// Library/Structures/Miscellaneous/RCSupportedFunctions
{attribute 'pack_mode' := '1'} 
// ------------------------------------------------------------------------- 
//  SRCI Robot Library                                                
// ------------------------------------------------------------------------- 
//                                                                           
//  Object:      RCSupportedFunctions                                       
//  Author:      Thorsten Brach                                                
//  Date:        2024-06-01
//
//  Description:                                              
//   
//                                                                           
//  Copyright: 
//    (C) 2024 Thorsten Brach. All rights reserved                                                                                                                                            
//             Licensed under the LGPL-3.0 license.
//                                                                           
//  Disclaimer:                                                                           
//    This project is provided without any guarantee and can be used for   
//    private and commercial purposes. Any use is at the user’s 
//    own risk and responsibility.
//
// -------------------------------------------------------------------------
TYPE RCSupportedFunctions :
STRUCT
  /// Byte 00 - Bit 0  
  Reserved                   : BOOL;
  /// Byte 00 - Bit 1 -> must be initialized with true, because this command is part of the interface initialization
  ReadRobotData              : BOOL := TRUE; 
  /// Byte 00 - Bit 2  
  EnableRobot                : BOOL;
  /// Byte 00 - Bit 3  
  GroupReset                 : BOOL;
  /// Byte 00 - Bit 4  
  ReadActualPosition         : BOOL;
  /// Byte 00 - Bit 5 
  ReadActualPositionCyclic   : BOOL;
  /// Byte 00 - Bit 6  -> must be initialized with true, because this command is part of the interface initialization
  ExchangeConfiguration      : BOOL := TRUE; 
  /// Byte 00 - Bit 7  
  SetSequence                : BOOL;
  
  /// Byte 01 - Bit 0  
  ChangeSpeedOverride        : BOOL;
  /// Byte 01 - Bit 1  ->  must be initialized with true, because this command is part of the interface initialization
  ReadMessages               : BOOL := TRUE; 
  /// Byte 01 - Bit 2  
  ReadRobotReferenceDynamics : BOOL;
  /// Byte 01 - Bit 3  
  WriteFrameData             : BOOL;
  /// Byte 01 - Bit 4  
  WriteToolData              : BOOL;
  /// Byte 01 - Bit 5  
  WriteLoadData              : BOOL;
  /// Byte 01 - Bit 6  
  WriteRobotReferenceDynamics: BOOL;
  /// Byte 01 - Bit 7  
  WriteRobotDefaultDynamics  : BOOL;
  
  /// Byte 02 - Bit 0  
  ReadRobotDefaultDynamics   : BOOL;
  /// Byte 02 - Bit 1  
  ReadFrameData              : BOOL;
  /// Byte 02 - Bit 2  
  ReadToolData               : BOOL;
  /// Byte 02 - Bit 3  
  ReadLoadData               : BOOL;
  /// Byte 02 - Bit 4  
  ReadRobotSWLimits          : BOOL;
  /// Byte 02 - Bit 5  
  GroupJog                   : BOOL;
  /// Byte 02 - Bit 6  
  MoveLinearAbsolute         : BOOL;
  /// Byte 02 - Bit 7  
  MoveDirectAbsolute         : BOOL;
  
  /// Byte 03 - Bit 0  
  MoveAxesAbsolute           : BOOL;
  /// Byte 03 - Bit 1  
  GroupStop                  : BOOL;
  /// Byte 03 - Bit 2
  GroupContinue              : BOOL;
  /// Byte 03 - Bit 3
  GroupInterrupt             : BOOL;
  /// Byte 03 - Bit 4
  ReturnToPrimary            : BOOL;
  /// Byte 03 - Bit 5
  MoveLinearAbsoluteJ        : BOOL;
  /// Byte 03 - Bit 6
  MoveDirectRelative         : BOOL;
  /// Byte 03 - Bit 7
  MoveAxesRelative           : BOOL;
  
  /// Byte 04 - Bit 0
  MoveCircularAbsolute       : BOOL;
  /// Byte 04 - Bit 1
  MoveCircularRelative       : BOOL;
  /// Byte 04 - Bit 2
  MoveLinearOffset           : BOOL;
  /// Byte 04 - Bit 3
  MoveDirectOffset           : BOOL;
  /// Byte 04 - Bit 4
  WaitTime                   : BOOL;
  /// Byte 04 - Bit 5
  ReadDigitalInputs          : BOOL;
  /// Byte 04 - Bit 6
  ReadDigitalOutputs         : BOOL;
  /// Byte 04 - Bit 7
  WriteDigitalOutputs        : BOOL;
  
  /// Byte 05 - Bit 0
  ReadIntegers               : BOOL;
  /// Byte 05 - Bit 1
  ReadReals                  : BOOL;
  /// Byte 05 - Bit 2
  WriteIntegers              : BOOL;
  /// Byte 05 - Bit 3
  WriteReals                 : BOOL;
  /// Byte 05 - Bit 4
  MoveLinearCam              : BOOL;
  /// Byte 05 - Bit 5
  MoveDirectCam              : BOOL;
  /// Byte 05 - Bit 6
  MoveCircularCam            : BOOL;
  /// Byte 05 - Bit 7
  SetTriggerRegister         : BOOL;
  
  /// Byte 06 - Bit 0
  SetTriggerLimit            : BOOL;
  /// Byte 06 - Bit 1
  SetTriggerUser             : BOOL;
  /// Byte 06 - Bit 2
  SetTriggerError            : BOOL;
  /// Byte 06 - Bit 3
  ReactAtTrigger             : BOOL;
  /// Byte 06 - Bit 4
  WaitForTrigger             : BOOL;
  /// Byte 06 - Bit 5
  ReadSystemVariable         : BOOL;
  /// Byte 06 - Bit 6
  WriteSystemVariable        : BOOL;
  /// Byte 06 - Bit 7
  CalculateForwardKinematic  : BOOL;
  
  /// Byte 07 - Bit 0
  CalculateInverseKinematic  : BOOL;
  /// Byte 07 - Bit 1
  CalculateCartesianPosition : BOOL;
  /// Byte 07 - Bit 2
  CalculateTool              : BOOL;
  /// Byte 07 - Bit 3
  CalculateFrame             : BOOL;
  /// Byte 07 - Bit 4
  ActivateNextCommand        : BOOL;
  /// Byte 07 - Bit 5
  ShiftPosition              : BOOL;
  /// Byte 07 - Bit 6
  CallSubprogram             : BOOL;
  /// Byte 07 - Bit 7
  MoveLinearRelative         : BOOL;
  
  /// Byte 08 - Bit 0
  WriteCallSubprogramCyclic  : BOOL;
  /// Byte 08 - Bit 1
  ReadCallSubprogramCyclic   : BOOL;
  /// Byte 08 - Bit 2
  StopSubprogram             : BOOL;
  /// Byte 08 - Bit 3
  ReadDHParameter            : BOOL;
  /// Byte 08 - Bit 4
  RestartController          : BOOL;
  /// Byte 08 - Bit 5
  ReadActualTCPVelocity      : BOOL;
  /// Byte 08 - Bit 6
  UserLogin                  : BOOL;
  /// Byte 08 - Bit 7
  SwitchLanguage             : BOOL;
  
  /// Byte 09 - Bit 0
  WriteRobotSWLimits         : BOOL;
  /// Byte 09 - Bit 1
  SetOperationMode           : BOOL;
  /// Byte 09 - Bit 2
  ReadWorkArea               : BOOL;
  /// Byte 09 - Bit 3
  WriteWorkArea              : BOOL;
  /// Byte 09 - Bit 4
  ActivateWorkArea           : BOOL;
  /// Byte 09 - Bit 5
  MonitorWorkArea            : BOOL;
  /// Byte 09 - Bit 6
  MoveApproachLinear         : BOOL;
  /// Byte 09 - Bit 7
  MoveDepartLinear           : BOOL;
  
  /// Byte 10 - Bit 0
  MoveApproachDirect         : BOOL;
  /// Byte 10 - Bit 1
  MoveDepartDirect           : BOOL;
  /// Byte 10 - Bit 2
  SearchHardstop             : BOOL;
  /// Byte 10 - Bit 3
  SearchHardstopJ            : BOOL;
  /// Byte 10 - Bit 4
  MovePickPlaceLinear        : BOOL;
  /// Byte 10 - Bit 5
  MovePickPlaceDirect        : BOOL;
  /// Byte 10 - Bit 6
  ActivateConveyorTracking   : BOOL;
  /// Byte 10 - Bit 7
  RedefineTrackingPosition   : BOOL;

  /// Byte 11 - Bit 0
  SyncToConveyor             : BOOL;
  /// Byte 11 - Bit 1
  ConfigureConveyor          : BOOL;
  /// Byte 11 - Bit 2
  MoveSuperImposed           : BOOL;
  /// Byte 11 - Bit 3
  MoveSuperImposedDynamic    : BOOL;
  /// Byte 11 - Bit 4
  ReadAnalogInput            : BOOL;
  /// Byte 11 - Bit 5
  ReadAnalogOutput           : BOOL;
  /// Byte 11 - Bit 6
  WriteAnalogOutput          : BOOL;
  /// Byte 11 - Bit 7
  MeasuringInput             : BOOL;

  /// Byte 12 - Bit 0
  AbortMeasuringInput        : BOOL;
  /// Byte 12 - Bit 1
  SetTriggerMotion           : BOOL;
  /// Byte 12 - Bit 2
  OpenBrake                  : BOOL;
  /// Byte 12 - Bit 3
  PathAccuracyMode           : BOOL;
  /// Byte 12 - Bit 4
  AvoidSingularity           : BOOL;
  /// Byte 12 - Bit 5
  ForceControl               : BOOL;
  /// Byte 12 - Bit 6
  ForceLimit                 : BOOL;
  /// Byte 12 - Bit 7
  ReadActualForce            : BOOL;
  
  /// Byte 13 - Bit 0
  BrakeTest                  : BOOL;
  /// Byte 13 - Bit 1
  SoftSwitchTCP              : BOOL;
  /// Byte 13 - Bit 2
  CreateSpline               : BOOL;
  /// Byte 13 - Bit 3
  DeleteSpline               : BOOL;
  /// Byte 13 - Bit 4
  MoveSpline                 : BOOL;
  /// Byte 13 - Bit 5
  DynamicSpline              : BOOL;
  /// Byte 13 - Bit 6
  LoadMeasurementAutomatic   : BOOL;
  /// Byte 13 - Bit 7
  LoadMeasurementSequential  : BOOL;
  
  /// Byte 14 - Bit 0
  CollisionDetection         : BOOL;
  /// Byte 14 - Bit 1
  FreeDrive                  : BOOL;
  /// Byte 14 - Bit 2
  UnitMeasurement            : BOOL;
  /// Byte 14 - Bit 3
  Byte14Bit03                : BOOL;
  /// Byte 14 - Bit 4
  Byte14Bit04                : BOOL;
  /// Byte 14 - Bit 5
  Byte14Bit05                : BOOL;
  /// Byte 14 - Bit 6
  Byte14Bit06                : BOOL;
  /// Byte 14 - Bit 7
  Byte14Bit07                : BOOL;
  
  /// Byte 15 - Bit 0
  Byte15Bit00                : BOOL;
  /// Byte 15 - Bit 1
  Byte15Bit01                : BOOL;
  /// Byte 15 - Bit 2
  Byte15Bit02                : BOOL;
  /// Byte 15 - Bit 3
  Byte15Bit03                : BOOL;
  /// Byte 15 - Bit 4
  Byte15Bit04                : BOOL;
  /// Byte 15 - Bit 5
  Byte15Bit05                : BOOL;
  /// Byte 15 - Bit 6
  Byte15Bit06                : BOOL;
  /// Byte 15 - Bit 7
  Byte15Bit07                : BOOL;

  /// Byte 16 - Bit 0
  Byte16Bit00                : BOOL;
  /// Byte 15 - Bit 1
  Byte16Bit01                : BOOL;
  /// Byte 15 - Bit 2
  Byte16Bit02                : BOOL;
  /// Byte 15 - Bit 3
  Byte16Bit03                : BOOL;
  /// Byte 15 - Bit 4
  Byte16Bit04                : BOOL;
  /// Byte 15 - Bit 5
  Byte16Bit05                : BOOL;
  /// Byte 15 - Bit 6
  Byte16Bit06                : BOOL;
  /// Byte 15 - Bit 7
  Byte16Bit07                : BOOL;
  
  /// Byte 17 - Bit 0
  Byte17Bit00                : BOOL;
  /// Byte 17 - Bit 1
  Byte17Bit01                : BOOL;
  /// Byte 17 - Bit 2
  Byte17Bit02                : BOOL;
  /// Byte 17 - Bit 3
  Byte17Bit03                : BOOL;
  /// Byte 17 - Bit 4
  Byte17Bit04                : BOOL;
  /// Byte 17 - Bit 5
  Byte17Bit05                : BOOL;
  /// Byte 17 - Bit 6
  Byte17Bit06                : BOOL;
  /// Byte 17 - Bit 7
  Byte17Bit07                : BOOL;

  /// Byte 18 - Bit 0
  Byte18Bit00                : BOOL;
  /// Byte 18 - Bit 1
  Byte18Bit01                : BOOL;
  /// Byte 18 - Bit 2
  Byte18Bit02                : BOOL;
  /// Byte 18 - Bit 3
  Byte18Bit03                : BOOL;
  /// Byte 18 - Bit 4
  Byte18Bit04                : BOOL;
  /// Byte 18 - Bit 5
  Byte18Bit05                : BOOL;
  /// Byte 18 - Bit 6
  Byte18Bit06                : BOOL;
  /// Byte 18 - Bit 7
  Byte18Bit07                : BOOL;
END_STRUCT
END_TYPE

// Library/Structures/Miscellaneous/RobotAxesFlags
{attribute 'pack_mode' := '1'} 
// ------------------------------------------------------------------------- 
//  SRCI Robot Library                                                
// ------------------------------------------------------------------------- 
//                                                                           
//  Object:      RobotAxesFlags                                       
//  Author:      Thorsten Brach                                                
//  Date:        2024-06-01
//
//  Description:                                              
//   
//                                                                           
//  Copyright: 
//    (C) 2024 Thorsten Brach. All rights reserved                                                                                                                                            
//             Licensed under the LGPL-3.0 license.
//                                                                           
//  Disclaimer:                                                                           
//    This project is provided without any guarantee and can be used for   
//    private and commercial purposes. Any use is at the user’s 
//    own risk and responsibility.
//
// -------------------------------------------------------------------------
TYPE RobotAxesFlags :
STRUCT
  /// Bit00 : Not used
  Bit00   : BOOL;
  /// Bit01 : Robot axis J1 - property depends of usage 
  AxisJ1  : BOOL;
  /// Bit02 : Robot axis J2 - property depends of usage 
  AxisJ2  : BOOL;
  /// Bit03 : Robot axis J3 - property depends of usage 
  AxisJ3  : BOOL;
  /// Bit04 : Robot axis J4 - property depends of usage 
  AxisJ4  : BOOL;
  /// Bit05 : Robot axis J5 - property depends of usage 
  AxisJ5  : BOOL;
  /// Bit06 : Robot axis J6 - property depends of usage 
  AxisJ6  : BOOL;
  /// Bit07 : Not used
  Bit07   : BOOL;
END_STRUCT
END_TYPE

// Library/Structures/Miscellaneous/SWLimits
{attribute 'pack_mode' := '1'} 
// ------------------------------------------------------------------------- 
//  SRCI Robot Library                                                
// ------------------------------------------------------------------------- 
//                                                                           
//  Object:      SWLimits                                       
//  Author:      Thorsten Brach                                                
//  Date:        2024-06-01
//
//  Description:                                              
//   
//                                                                           
//  Copyright: 
//    (C) 2024 Thorsten Brach. All rights reserved                                                                                                                                            
//             Licensed under the LGPL-3.0 license.
//                                                                           
//  Disclaimer:                                                                           
//    This project is provided without any guarantee and can be used for   
//    private and commercial purposes. Any use is at the user’s 
//    own risk and responsibility.
//
// -------------------------------------------------------------------------
TYPE SWLimits :
STRUCT
  /// Timestamp
  Timestamp    : IEC_TIMESTAMP;
  /// Negative software limit for Joint J1 [mm/°]
  J1LowerLimit : REAL;
  /// Positive software limit for Joint J1 [mm/°]
  J1UpperLimit : REAL;
  /// Negative software limit for Joint J2 [mm/°]
  J2LowerLimit : REAL;
  /// Positive software limit for Joint J2 [mm/°]
  J2UpperLimit : REAL;
  /// Negative software limit for Joint J3 [mm/°]
  J3LowerLimit : REAL;
  /// Positive software limit for Joint J3 [mm/°]
  J3UpperLimit : REAL;
  /// Negative software limit for Joint J4 [mm/°]
  J4LowerLimit : REAL;
  /// Positive software limit for Joint J4 [mm/°]
  J4UpperLimit : REAL;
  /// Negative software limit for Joint J5 [mm/°]
  J5LowerLimit : REAL;
  /// Positive software limit for Joint J5 [mm/°]
  J5UpperLimit : REAL;
  /// Negative software limit for Joint J6 [mm/°]
  J6LowerLimit : REAL;
  /// Positive software limit for Joint J6 [mm/°]
  J6UpperLimit : REAL;
  /// Negative software limit for axis E1 [mm/°]
  E1LowerLimit : REAL;
  /// Positive software limit for axis E1 [mm/°]
  E1UpperLimit : REAL;
  /// Negative software limit for axis E2 [mm/°]
  E2LowerLimit : REAL;
  /// Positive software limit for axis E2 [mm/°]
  E2UpperLimit : REAL;
  /// Negative software limit for axis E3 [mm/°]
  E3LowerLimit : REAL;
  /// Positive software limit for axis E3 [mm/°]
  E3UpperLimit : REAL;
  /// Negative software limit for axis E4 [mm/°]
  E4LowerLimit : REAL;
  /// Positive software limit for axis E4 [mm/°]
  E4UpperLimit : REAL;
  /// Negative software limit for axis E5 [mm/°]
  E5LowerLimit : REAL;
  /// Positive software limit for axis E5 [mm/°]
  E5UpperLimit : REAL;
  /// Negative software limit for axis E6 [mm/°]
  E6LowerLimit : REAL;
  /// Positive software limit for axis E6 [mm/°]
  E6UpperLimit : REAL;  
END_STRUCT
END_TYPE

// Library/Structures/Miscellaneous/SynchronizationModes
{attribute 'pack_mode' := '1'} 
// ------------------------------------------------------------------------- 
//  SRCI Robot Library                                                
// ------------------------------------------------------------------------- 
//                                                                           
//  Object:      SynchronizationModes                                       
//  Author:      Thorsten Brach                                                
//  Date:        2024-06-01
//
//  Description:                                              
//   
//                                                                           
//  Copyright: 
//    (C) 2024 Thorsten Brach. All rights reserved                                                                                                                                            
//             Licensed under the LGPL-3.0 license.
//                                                                           
//  Disclaimer:                                                                           
//    This project is provided without any guarantee and can be used for   
//    private and commercial purposes. Any use is at the user’s 
//    own risk and responsibility.
//
// -------------------------------------------------------------------------
TYPE SynchronizationModes :
STRUCT
 /// synchronization direction for tool
 Tool              : SyncMode;
 /// synchronization direction for frame
 Frame             : SyncMode;
 /// synchronization direction for load
 Load              : SyncMode;
 /// synchronization direction for work areas
 WorkAreas         : SyncMode;
 /// synchronization direction for SW limits
 SWLimits          : SyncMode;
 /// synchronization direction for defaul dynamics
 DefaultDynamics   : SyncMode;
 /// synchronization direction for reference dynamics 
 ReferenceDynamics : SyncMode; 
END_STRUCT
END_TYPE

// Library/Structures/Miscellaneous/TrackingStatus
{attribute 'pack_mode' := '1'} 
// ------------------------------------------------------------------------- 
//  SRCI Robot Library                                                
// ------------------------------------------------------------------------- 
//                                                                           
//  Object:      TrackingStatus                                       
//  Author:      Thorsten Brach                                                
//  Date:        2024-06-01
//
//  Description:                                              
//   
//                                                                           
//  Copyright: 
//    (C) 2024 Thorsten Brach. All rights reserved                                                                                                                                            
//             Licensed under the LGPL-3.0 license.
//                                                                           
//  Disclaimer:                                                                           
//    This project is provided without any guarantee and can be used for   
//    private and commercial purposes. Any use is at the user’s 
//    own risk and responsibility.
//
// -------------------------------------------------------------------------
TYPE TrackingStatus :
STRUCT
  /// TRUE, while a "ConveyorTracking" function is enabled
  ConveyorTrackingEnabled   : BOOL;  
  /// TRUE, while robot is waiting for condition defined by "SyncInMode" after "SyncToConveyor" has been executed
  WaitingForSynchronization : BOOL;
  /// TRUE, while robot is matching the TCP’s velocity to the conveyor’s velocity
  Synchronizing             : BOOL;
  /// TRUE, while TCP is moving synchronously to conveyor
  Synchronous               : BOOL;
  /// TRUE, while robot is terminating synchronous movement
  Desynchronizing           : BOOL;
  /// TRUE, while assigned UCS is within "SyncOutZone"
  SyncOutZoneEntered        : BOOL;
  /// TRUE, when assigned UCS leaves "SyncOutZone"
  /// Reset, when robot’s synchronous movement has been stopped
  SyncOutZoneLeft           : BOOL;
  /// Not used
  NotUsed                   : BOOL;   
END_STRUCT
END_TYPE

// Library/Structures/Miscellaneous/TurnNumber
{attribute 'pack_mode' := '1'} 
// ------------------------------------------------------------------------- 
//  SRCI Robot Library                                                
// ------------------------------------------------------------------------- 
//                                                                           
//  Object:      TurnNumber                                       
//  Author:      Thorsten Brach                                                
//  Date:        2024-06-01
//
//  Description:                                              
//   
//                                                                           
//  Copyright: 
//    (C) 2024 Thorsten Brach. All rights reserved                                                                                                                                            
//             Licensed under the LGPL-3.0 license.
//                                                                           
//  Disclaimer:                                                                           
//    This project is provided without any guarantee and can be used for   
//    private and commercial purposes. Any use is at the user’s 
//    own risk and responsibility.
//
// -------------------------------------------------------------------------
TYPE TurnNumber :
STRUCT
  /// Turn number of J1
  J1Turns : SINT;
  /// Turn number of J2
  J2Turns : SINT;
  /// Turn number of J3
  J3Turns : SINT;
  /// Turn number of J4
  J4Turns : SINT;
  /// Turn number of J5
  J5Turns : SINT;
  /// Turn number of J6
  J6Turns : SINT;
  /// Turn number of E1
  E1Turns : SINT;  
END_STRUCT
END_TYPE

// Library/Structures/Miscellaneous/VersionStruct
{attribute 'pack_mode' := '1'} 
// ------------------------------------------------------------------------- 
//  SRCI Robot Library                                                
// ------------------------------------------------------------------------- 
//                                                                           
//  Object:      VersionStruct                                       
//  Author:      Thorsten Brach                                                
//  Date:        2024-06-01
//
//  Description:                                              
//   
//                                                                           
//  Copyright: 
//    (C) 2024 Thorsten Brach. All rights reserved                                                                                                                                            
//             Licensed under the LGPL-3.0 license.
//                                                                           
//  Disclaimer:                                                                           
//    This project is provided without any guarantee and can be used for   
//    private and commercial purposes. Any use is at the user’s 
//    own risk and responsibility.
//
// -------------------------------------------------------------------------
TYPE VersionStruct :
STRUCT
  /// Major version
  MajorVersion : USINT;
  /// Minor version
  MinorVersion : USINT;
  /// Patch version  
  PatchVersion : USINT;
END_STRUCT
END_TYPE

// Library/Structures/Telegram/PlcToRob/Command/TelegramPlcToRobCommand
{attribute 'pack_mode' := '1'} 
// ------------------------------------------------------------------------- 
//  SRCI Robot Library                                                
// ------------------------------------------------------------------------- 
//                                                                           
//  Object:      TelegramPlcToRobMessage                                       
//  Author:      Thorsten Brach                                                
//  Date:        2024-06-01
//
//  Description:                                              
//   
//                                                                           
//  Copyright: 
//    (C) 2024 Thorsten Brach. All rights reserved                                                                                                                                            
//             Licensed under the LGPL-3.0 license.
//                                                                           
//  Disclaimer:                                                                           
//    This project is provided without any guarantee and can be used for   
//    private and commercial purposes. Any use is at the user’s 
//    own risk and responsibility.
//
// -------------------------------------------------------------------------
TYPE TelegramPlcToRobCommand :
STRUCT
  /// Header
  Header  : TelegramPlcToRobCommandHeader;
  /// Payload
  Payload : ARRAY[0..255] OF BYTE; // ToDo
END_STRUCT
END_TYPE

// Library/Structures/Telegram/PlcToRob/Command/TelegramPlcToRobCommandHeader
{attribute 'pack_mode' := '1'} 
// ------------------------------------------------------------------------- 
//  SRCI Robot Library                                                
// ------------------------------------------------------------------------- 
//                                                                           
//  Object:      TelegramPlcToRobMessageHeader                                       
//  Author:      Thorsten Brach                                                
//  Date:        2024-06-01
//
//  Description:                                              
//   
//                                                                           
//  Copyright: 
//    (C) 2024 Thorsten Brach. All rights reserved                                                                                                                                            
//             Licensed under the LGPL-3.0 license.
//                                                                           
//  Disclaimer:                                                                           
//    This project is provided without any guarantee and can be used for   
//    private and commercial purposes. Any use is at the user’s 
//    own risk and responsibility.
//
// -------------------------------------------------------------------------
TYPE TelegramPlcToRobCommandHeader :
STRUCT
  /// Command type
  CmdType           : CmdType;
  /// CMD priority level
  Prio              : PriorityLevel;
  /// Execution Mode
  ExecMode          : ExecutionMode;
  /// Parameter Sequence
  ParSequence       : BYTE;
END_STRUCT
END_TYPE

// Library/Structures/Telegram/PlcToRob/Cyclic/TelegramPlcToRobCyclicData
{attribute 'pack_mode' := '1'} 
// ------------------------------------------------------------------------- 
//  SRCI Robot Library                                                
// ------------------------------------------------------------------------- 
//                                                                           
//  Object:      TelegramPlcToRobCyclicData                                       
//  Author:      Thorsten Brach                                                
//  Date:        2024-11-30
//
//  Description:                                              
//   
//                                                                           
//  Copyright: 
//    (C) 2024 Thorsten Brach. All rights reserved                                                                                                                                            
//             Licensed under the LGPL-3.0 license.
//                                                                           
//  Disclaimer:                                                                           
//    This project is provided without any guarantee and can be used for   
//    private and commercial purposes. Any use is at the user’s 
//    own risk and responsibility.
//
// -------------------------------------------------------------------------
TYPE TelegramPlcToRobCyclicData :
STRUCT
  /// Current Tool
  ToolNo  : BYTE;
  /// Current Frame
  FrameNo : BYTE;      
END_STRUCT
END_TYPE

// Library/Structures/Telegram/PlcToRob/CyclicOptional/Internal/TelegramPlcToRobCyclicOptionalCartesianPosition
{attribute 'pack_mode' := '1'} 
// ------------------------------------------------------------------------- 
//  SRCI Robot Library                                                
// ------------------------------------------------------------------------- 
//                                                                           
//  Object:      TelegramPlcToRobCyclicOptionalCartesianPos                                       
//  Author:      Thorsten Brach                                                
//  Date:        2024-06-01
//
//  Description:                                              
//   
//                                                                           
//  Copyright: 
//    (C) 2024 Thorsten Brach. All rights reserved                                                                                                                                            
//             Licensed under the LGPL-3.0 license.
//                                                                           
//  Disclaimer:                                                                           
//    This project is provided without any guarantee and can be used for   
//    private and commercial purposes. Any use is at the user’s 
//    own risk and responsibility.
//
// -------------------------------------------------------------------------
TYPE TelegramPlcToRobCyclicOptionalCartesianPosition :
STRUCT
  /// TCP Position on the X-Axis
  X           : REAL;
  /// TCP Position on the Y-Axis
  Y           : REAL;
  /// TCP Position on the Z-Axis
  Z           : REAL;
  /// Rotation around the X-Axis (RX)
  Rx          : REAL;
  /// Rotation around the Y-Axis (RY)
  Ry          : REAL;
  /// Rotation around the Z-Axis (RZ)
  Rz          : REAL;
  /// Configuration
  Config      : WORD;
  /// Turns of J1 and J2
  Turns_J2_J1 : BYTE;
  /// Turns of J3 and J4
  Turns_J4_J3 : BYTE;
  /// Turns of J6 and J5
  Turns_J6_J5 : BYTE;
  /// Turns of E1
  Turns_E1    : BYTE;
  /// Position of first external axis
  E1          : REAL;
END_STRUCT
END_TYPE

// Library/Structures/Telegram/PlcToRob/CyclicOptional/Internal/TelegramPlcToRobCyclicOptionalCartesianPositionExt
{attribute 'pack_mode' := '1'} 
// ------------------------------------------------------------------------- 
//  SRCI Robot Library                                                
// ------------------------------------------------------------------------- 
//                                                                           
//  Object:      TelegramPlcToRobCyclicOptionalCartesianPositionExt                                       
//  Author:      Thorsten Brach                                                
//  Date:        2024-06-01
//
//  Description:                                              
//   
//                                                                           
//  Copyright: 
//    (C) 2024 Thorsten Brach. All rights reserved                                                                                                                                            
//             Licensed under the LGPL-3.0 license.
//                                                                           
//  Disclaimer:                                                                           
//    This project is provided without any guarantee and can be used for   
//    private and commercial purposes. Any use is at the user’s 
//    own risk and responsibility.
//
// -------------------------------------------------------------------------
TYPE TelegramPlcToRobCyclicOptionalCartesianPositionExt :
STRUCT
  /// Position of second external axis
  E2 : REAL;
  /// Position of third external axis
  E3 : REAL;
  /// Position of fourth external axis
  E4 : REAL;
  /// Position of fifth external axis
  E5 : REAL;
  /// Position of sixth external axis
  E6 : REAL;    
END_STRUCT
END_TYPE

// Library/Structures/Telegram/PlcToRob/CyclicOptional/Internal/TelegramPlcToRobCyclicOptionalCurrent
{attribute 'pack_mode' := '1'} 
// ------------------------------------------------------------------------- 
//  SRCI Robot Library                                                
// ------------------------------------------------------------------------- 
//                                                                           
//  Object:      TelegramPlcToRobCyclicOptionalCurrent                                       
//  Author:      Thorsten Brach                                                
//  Date:        2024-06-01
//
//  Description:                                              
//   
//                                                                           
//  Copyright: 
//    (C) 2024 Thorsten Brach. All rights reserved                                                                                                                                            
//             Licensed under the LGPL-3.0 license.
//                                                                           
//  Disclaimer:                                                                           
//    This project is provided without any guarantee and can be used for   
//    private and commercial purposes. Any use is at the user’s 
//    own risk and responsibility.
//
// -------------------------------------------------------------------------
TYPE TelegramPlcToRobCyclicOptionalCurrent :
STRUCT
  /// Current of first joint of the robot
  J1 : REAL;
  /// Current of second joint of the robot
  J2 : REAL;
  /// Current of third joint of the robot
  J3 : REAL;
  /// Current of fourth joint of the robot
  J4 : REAL;
  /// Current of fifth joint of the robot
  J5 : REAL;
  /// Current of sixth joint of the robot
  J6 : REAL;  
END_STRUCT
END_TYPE

// Library/Structures/Telegram/PlcToRob/CyclicOptional/Internal/TelegramPlcToRobCyclicOptionalCurrentExt
{attribute 'pack_mode' := '1'} 
// ------------------------------------------------------------------------- 
//  SRCI Robot Library                                                
// ------------------------------------------------------------------------- 
//                                                                           
//  Object:      TelegramPlcToRobCyclicOptionalCurrentExt                                       
//  Author:      Thorsten Brach                                                
//  Date:        2024-06-01
//
//  Description:                                              
//   
//                                                                           
//  Copyright: 
//    (C) 2024 Thorsten Brach. All rights reserved                                                                                                                                            
//             Licensed under the LGPL-3.0 license.
//                                                                           
//  Disclaimer:                                                                           
//    This project is provided without any guarantee and can be used for   
//    private and commercial purposes. Any use is at the user’s 
//    own risk and responsibility.
//
// -------------------------------------------------------------------------
TYPE TelegramPlcToRobCyclicOptionalCurrentExt :
STRUCT
  /// Current of first external joint of the robot
  E1 : REAL;
  /// Current of second external axis
  E2: REAL;
  /// Current of third external axis
  E3: REAL;
  /// Current of fourth external axis
  E4: REAL;
  /// Current of fifth external axis
  E5: REAL;
  /// Current of sixth external axis
  E6: REAL;  
END_STRUCT
END_TYPE

// Library/Structures/Telegram/PlcToRob/CyclicOptional/Internal/TelegramPlcToRobCyclicOptionalForce
{attribute 'pack_mode' := '1'} 
// ------------------------------------------------------------------------- 
//  SRCI Robot Library                                                
// ------------------------------------------------------------------------- 
//                                                                           
//  Object:      TelegramPlcToRobCyclicOptionalForce                                       
//  Author:      Thorsten Brach                                                
//  Date:        2024-06-01
//
//  Description:                                              
//   
//                                                                           
//  Copyright: 
//    (C) 2024 Thorsten Brach. All rights reserved                                                                                                                                            
//             Licensed under the LGPL-3.0 license.
//                                                                           
//  Disclaimer:                                                                           
//    This project is provided without any guarantee and can be used for   
//    private and commercial purposes. Any use is at the user’s 
//    own risk and responsibility.
//
// -------------------------------------------------------------------------
TYPE TelegramPlcToRobCyclicOptionalForce :
STRUCT
  /// Force on the X-Axis
  X : REAL;
  /// Force on the Y-Axis
  Y : REAL;
  /// Force on the Z-Axis
  Z : REAL;
  /// Force around the X-Axis (RX)
  Rx : REAL;
  /// Force around the Y-Axis (RY)
  Ry : REAL;
  /// Force around the Z-Axis (RZ)
  Rz : REAL;
END_STRUCT
END_TYPE

// Library/Structures/Telegram/PlcToRob/CyclicOptional/Internal/TelegramPlcToRobCyclicOptionalForceExt
{attribute 'pack_mode' := '1'} 
// ------------------------------------------------------------------------- 
//  SRCI Robot Library                                                
// ------------------------------------------------------------------------- 
//                                                                           
//  Object:      TelegramPlcToRobCyclicOptionalForceExt                                       
//  Author:      Thorsten Brach                                                
//  Date:        2024-06-01
//
//  Description:                                              
//   
//                                                                           
//  Copyright: 
//    (C) 2024 Thorsten Brach. All rights reserved                                                                                                                                            
//             Licensed under the LGPL-3.0 license.
//                                                                           
//  Disclaimer:                                                                           
//    This project is provided without any guarantee and can be used for   
//    private and commercial purposes. Any use is at the user’s 
//    own risk and responsibility.
//
// -------------------------------------------------------------------------
TYPE TelegramPlcToRobCyclicOptionalForceExt :
STRUCT
  /// Force on the external axis 1
  E1 : REAL;
  /// Force on the external axis 2
  E2 : REAL;
  /// Force on the external axis 3
  E3 : REAL;
  /// Force om the external axis 4
  E4 : REAL;
  /// Force on the external axis 5
  E5 : REAL;
  /// Force on the external axis 6
  E6 : REAL;
END_STRUCT
END_TYPE

// Library/Structures/Telegram/PlcToRob/CyclicOptional/Internal/TelegramPlcToRobCyclicOptionalJointPosition
{attribute 'pack_mode' := '1'} 
// ------------------------------------------------------------------------- 
//  SRCI Robot Library                                                
// ------------------------------------------------------------------------- 
//                                                                           
//  Object:      TelegramPlcToRobCyclicOptionalJointPosition                                       
//  Author:      Thorsten Brach                                                
//  Date:        2024-06-01
//
//  Description:                                              
//   
//                                                                           
//  Copyright: 
//    (C) 2024 Thorsten Brach. All rights reserved                                                                                                                                            
//             Licensed under the LGPL-3.0 license.
//                                                                           
//  Disclaimer:                                                                           
//    This project is provided without any guarantee and can be used for   
//    private and commercial purposes. Any use is at the user’s 
//    own risk and responsibility.
//
// -------------------------------------------------------------------------
TYPE TelegramPlcToRobCyclicOptionalJointPosition :
STRUCT
  /// Position of first joint of the robot
  J1 : REAL;
  /// Position of second joint of the robot
  J2 : REAL;
  /// Position of third joint of the robot
  J3 : REAL;
  /// Position of fourth joint of the robot
  J4 : REAL;
  /// Position of fifth joint of the robot
  J5 : REAL;
  /// Position of sixth joint of the robot
  J6 : REAL;
  /// Position of first external axis 
  E1 : REAL;  
END_STRUCT
END_TYPE

// Library/Structures/Telegram/PlcToRob/CyclicOptional/Internal/TelegramPlcToRobCyclicOptionalJointPositionExt
{attribute 'pack_mode' := '1'} 
// ------------------------------------------------------------------------- 
//  SRCI Robot Library                                                
// ------------------------------------------------------------------------- 
//                                                                           
//  Object:      TelegramPlcToRobCyclicOptionalJointPositionExt                                       
//  Author:      Thorsten Brach                                                
//  Date:        2024-06-01
//
//  Description:                                              
//   
//                                                                           
//  Copyright: 
//    (C) 2024 Thorsten Brach. All rights reserved                                                                                                                                            
//             Licensed under the LGPL-3.0 license.
//                                                                           
//  Disclaimer:                                                                           
//    This project is provided without any guarantee and can be used for   
//    private and commercial purposes. Any use is at the user’s 
//    own risk and responsibility.
//
// -------------------------------------------------------------------------
TYPE TelegramPlcToRobCyclicOptionalJointPositionExt :
STRUCT
  /// Position of second external axis
  E2: REAL;
  /// Position of third external axis
  E3: REAL;
  /// Position of fourth external axis
  E4: REAL;
  /// Position of fifth external axis
  E5: REAL;
  /// Position of sixth external axis
  E6: REAL;    
END_STRUCT
END_TYPE

// Library/Structures/Telegram/PlcToRob/CyclicOptional/Internal/TelegramPlcToRobCyclicOptionalSubProgramData
{attribute 'pack_mode' := '1'} 
// ------------------------------------------------------------------------- 
//  SRCI Robot Library                                                
// ------------------------------------------------------------------------- 
//                                                                           
//  Object:      TelegramPlcToRobCyclicOptionalSubProgramData                                       
//  Author:      Thorsten Brach                                                
//  Date:        2024-06-01
//
//  Description:                                              
//   
//                                                                           
//  Copyright: 
//    (C) 2024 Thorsten Brach. All rights reserved                                                                                                                                            
//             Licensed under the LGPL-3.0 license.
//                                                                           
//  Disclaimer:                                                                           
//    This project is provided without any guarantee and can be used for   
//    private and commercial purposes. Any use is at the user’s 
//    own risk and responsibility.
//
// -------------------------------------------------------------------------
TYPE TelegramPlcToRobCyclicOptionalSubProgramData :
STRUCT
  /// Sub program data
  Data : ARRAY [0..25] OF BYTE;
END_STRUCT
END_TYPE

// Library/Structures/Telegram/PlcToRob/CyclicOptional/TelegramPlcToRobCyclicOptionalData
{attribute 'pack_mode' := '1'} 
// ------------------------------------------------------------------------- 
//  SRCI Robot Library                                                
// ------------------------------------------------------------------------- 
//                                                                           
//  Object:      TelegramPlcToRobCyclicOptionalData                                       
//  Author:      Thorsten Brach                                                
//  Date:        2024-06-01
//
//  Description:                                              
//   
//                                                                           
//  Copyright: 
//    (C) 2024 Thorsten Brach. All rights reserved                                                                                                                                            
//             Licensed under the LGPL-3.0 license.
//                                                                           
//  Disclaimer:                                                                           
//    This project is provided without any guarantee and can be used for   
//    private and commercial purposes. Any use is at the user’s 
//    own risk and responsibility.
//
// -------------------------------------------------------------------------
TYPE TelegramPlcToRobCyclicOptionalData :
STRUCT
  /// Transmit cyclic data from PLC to RC for the usage in a subprogram on the RC called via the function “CallSubprogram”
  SubProgramData        :  TelegramPlcToRobCyclicOptionalSubProgramData;
  /// short cartesian position with TCP position (X, Y,Z), rotation (RX, RY, RZ), configuration bytes (Config, TurnNumber), position of first external axis (E1) and corresponding coordinate systems (ToolNo, FrameNo)
  CartesianPosition     :  TelegramPlcToRobCyclicOptionalCartesianPosition;
  /// the external axis values for an extended cartesian position (E2, E3, E4, E5, E6) 
  /// When selected, Tool and Frame will automatically cyclically be sent from client to server.
  CartesianPositionExt  :  TelegramPlcToRobCyclicOptionalCartesianPositionExt;
  /// short axes position with joint values (J1, J2, J3,J4, J5, J6) and position of first external axis (E1)
  JointPosition         :  TelegramPlcToRobCyclicOptionalJointPosition;
  /// the external axis values for an extended joint position (E2, E3, E4, E5, E6)
  JointPositionExt      :  TelegramPlcToRobCyclicOptionalJointPositionExt;
  /// force with the divided forces in the individual directions (X, Y, Z, RX, RY, RZ)
  Force                 :  TelegramPlcToRobCyclicOptionalForce;
  /// current force for the external axis (E1, E2, E3, E4, E5, E6)
  ForceExt              :  TelegramPlcToRobCyclicOptionalForceExt;
  /// ctual axes current of individual axes (J1, J2, J3, J4, J5, J6)
  Current               :  TelegramPlcToRobCyclicOptionalCurrent;
  /// actual current for the external axis (E1, E2,E3, E4, E5, E6)
  CurrentExt            :  TelegramPlcToRobCyclicOptionalCurrentExt;
END_STRUCT
END_TYPE

// Library/Structures/Telegram/PlcToRob/Footer/TelegramPlcToRobFooter
{attribute 'pack_mode' := '1'} 
// ------------------------------------------------------------------------- 
//  SRCI Robot Library                                                
// ------------------------------------------------------------------------- 
//                                                                           
//  Object:      TelegramPlcToRobFooter                                       
//  Author:      Thorsten Brach                                                
//  Date:        2024-06-01
//
//  Description:                                              
//   
//                                                                           
//  Copyright: 
//    (C) 2024 Thorsten Brach. All rights reserved                                                                                                                                            
//             Licensed under the LGPL-3.0 license.
//                                                                           
//  Disclaimer:                                                                           
//    This project is provided without any guarantee and can be used for   
//    private and commercial purposes. Any use is at the user’s 
//    own risk and responsibility.
//
// -------------------------------------------------------------------------
TYPE TelegramPlcToRobFooter :
STRUCT
  /// Life Sign
  LifeSign : BYTE;
  /// Reserve
  Reserve  : BYTE;
END_STRUCT
END_TYPE

// Library/Structures/Telegram/PlcToRob/Fragment/TelegramPlcToRobFragment
{attribute 'pack_mode' := '1'} 
// ------------------------------------------------------------------------- 
//  SRCI Robot Library                                                
// ------------------------------------------------------------------------- 
//                                                                           
//  Object:      TelegramPlcToRobFragment                                       
//  Author:      Thorsten Brach                                                
//  Date:        2024-06-01
//
//  Description:                                              
//   
//                                                                           
//  Copyright: 
//    (C) 2024 Thorsten Brach. All rights reserved                                                                                                                                            
//             Licensed under the LGPL-3.0 license.
//                                                                           
//  Disclaimer:                                                                           
//    This project is provided without any guarantee and can be used for   
//    private and commercial purposes. Any use is at the user’s 
//    own risk and responsibility.
//
// -------------------------------------------------------------------------
TYPE TelegramPlcToRobFragment :
STRUCT
  /// Header
  Header  : TelegramPlcToRobFragmentHeader;
  /// Command
  Command : TelegramPlcToRobCommand;
END_STRUCT
END_TYPE

// Library/Structures/Telegram/PlcToRob/Fragment/TelegramPlcToRobFragmentHeader
{attribute 'pack_mode' := '1'} 
// ------------------------------------------------------------------------- 
//  SRCI Robot Library                                                
// ------------------------------------------------------------------------- 
//                                                                           
//  Object:      TelegramPlcToRobFragmentHeader                                       
//  Author:      Thorsten Brach                                                
//  Date:        2024-06-01
//
//  Description:                                              
//   
//                                                                           
//  Copyright: 
//    (C) 2024 Thorsten Brach. All rights reserved                                                                                                                                            
//             Licensed under the LGPL-3.0 license.
//                                                                           
//  Disclaimer:                                                                           
//    This project is provided without any guarantee and can be used for   
//    private and commercial purposes. Any use is at the user’s 
//    own risk and responsibility.
//
// -------------------------------------------------------------------------
TYPE TelegramPlcToRobFragmentHeader :
STRUCT
  /// Command Instance Identifier used to assign the CMD payload to a specific CMD instance
  CmdID          : UINT;
  /// Empty reserve byte
  Reserve        : BYTE;
  /// Fragment Action Byte
  FragmentAction : BYTE;
  /// Append received payload in the receive buffer at this position
  PayloadPointer : UINT;
  /// Length of the CMD payload
  PayloadLength  : UINT;  
END_STRUCT
END_TYPE

// Library/Structures/Telegram/PlcToRob/Header/TelegramPlcToRobHeader
{attribute 'pack_mode' := '1'} 
// ------------------------------------------------------------------------- 
//  SRCI Robot Library                                                
// ------------------------------------------------------------------------- 
//                                                                           
//  Object:      TelegramPlcToRobHeader                                       
//  Author:      Thorsten Brach                                                
//  Date:        2024-06-01
//
//  Description:                                              
//   
//                                                                           
//  Copyright: 
//    (C) 2024 Thorsten Brach. All rights reserved                                                                                                                                            
//             Licensed under the LGPL-3.0 license.
//                                                                           
//  Disclaimer:                                                                           
//    This project is provided without any guarantee and can be used for   
//    private and commercial purposes. Any use is at the user’s 
//    own risk and responsibility.
//
// -------------------------------------------------------------------------
TYPE TelegramPlcToRobHeader :
STRUCT
  /// Version of SRCI specification
  /// Bit 0-4 : Minor version = Features        (0..31)
  /// Bit 5-7 : Major version = Breaking change (0..07)
  SRCIVersion            : BYTE;
  /// Fast stop trigger | LifeSign
  FastStop_LifeSign      : BYTE;
  /// Number of Bytes of the frame to be used for the telegram of the given Axisgroup. Direction client to server
  TelegramLengthPlcToRob : UINT;
  /// Number of Bytes of the frame to be used for the telegram of the given Axisgroup. Direction server to client
  TelegramLengthRobToPlc : UINT;
  /// Control AxesGroupID | Telegtam state control
  AxesGroupID_Control    : BYTE;
  /// Reserved for later versions
  Reserved               : BYTE;
  /// Configuration of the optional cyclic data. Direction client to server
  TelegramNumberPlcToRob : UINT;
  /// Configuration of the optional cyclic data. Direction server to client
  TelegramNumberRobToPlc : UINT;
  /// Date of the client in the format days since 1990.01.01
  ClientDate             : IEC_DATE;
  /// Time in the clients time zone in the format milliseconds since start of day
  ClientTime             : IEC_TIME;  
END_STRUCT
END_TYPE

// Library/Structures/Telegram/PlcToRob/Sequence/TelegramPlcToRobSequence
{attribute 'pack_mode' := '1'} 
// ------------------------------------------------------------------------- 
//  SRCI Robot Library                                                
// ------------------------------------------------------------------------- 
//                                                                           
//  Object:      TelegramPlcToRobSequence                                       
//  Author:      Thorsten Brach                                                
//  Date:        2024-06-01
//
//  Description:                                              
//   
//                                                                           
//  Copyright: 
//    (C) 2024 Thorsten Brach. All rights reserved                                                                                                                                            
//             Licensed under the LGPL-3.0 license.
//                                                                           
//  Disclaimer:                                                                           
//    This project is provided without any guarantee and can be used for   
//    private and commercial purposes. Any use is at the user’s 
//    own risk and responsibility.
//
// -------------------------------------------------------------------------
TYPE TelegramPlcToRobSequence :
STRUCT
  /// Header
  Header   : TelegramPlcTorobSequenceHeader;
  /// Fragment
  Fragment : ARRAY[0..9] OF TelegramPlcToRobFragment;
END_STRUCT
END_TYPE

// Library/Structures/Telegram/PlcToRob/Sequence/TelegramPlcToRobSequenceHeader
{attribute 'pack_mode' := '1'} 
// ------------------------------------------------------------------------- 
//  SRCI Robot Library                                                
// ------------------------------------------------------------------------- 
//                                                                           
//  Object:      TelegramPlcTorobSequenceHeader                                       
//  Author:      Thorsten Brach                                                
//  Date:        2024-06-01
//
//  Description:                                              
//   
//                                                                           
//  Copyright: 
//    (C) 2024 Thorsten Brach. All rights reserved                                                                                                                                            
//             Licensed under the LGPL-3.0 license.
//                                                                           
//  Disclaimer:                                                                           
//    This project is provided without any guarantee and can be used for   
//    private and commercial purposes. Any use is at the user’s 
//    own risk and responsibility.
//
// -------------------------------------------------------------------------
TYPE TelegramPlcToRobSequenceHeader :
STRUCT
  /// Telegram Sequence and Acknowledgement number
  SEQ_ACK      : UINT;
  /// Length of the Telegram Sequence excluding this Telegram Sequence Header
  PayloadLength : UINT;
END_STRUCT
END_TYPE

// Library/Structures/Telegram/PlcToRob/TelegramPlcToRob
{attribute 'pack_mode' := '1'} 
// ------------------------------------------------------------------------- 
//  SRCI Robot Library                                                
// ------------------------------------------------------------------------- 
//                                                                           
//  Object:      TelegramPlcToRob                                       
//  Author:      Thorsten Brach                                                
//  Date:        2024-06-01
//
//  Description:                                              
//   
//                                                                           
//  Copyright: 
//    (C) 2024 Thorsten Brach. All rights reserved                                                                                                                                            
//             Licensed under the LGPL-3.0 license.
//                                                                           
//  Disclaimer:                                                                           
//    This project is provided without any guarantee and can be used for   
//    private and commercial purposes. Any use is at the user’s 
//    own risk and responsibility.
//
// -------------------------------------------------------------------------
TYPE TelegramPlcToRob :
STRUCT
  /// Header
  Header         : TelegramPlcToRobHeader;
  /// Cyclic optional data
  Cyclic         : TelegramPlcToRobCyclicData;
  /// Cyclic optional data
  CyclicOptional : TelegramPlcToRobCyclicOptionalData;
  /// Sequence Data
  Sequence       : ARRAY[0..1] OF TelegramPlcToRobSequence;
  /// Footer
  Footer         : TelegramPlcToRobFooter;
END_STRUCT
END_TYPE

// Library/Structures/Telegram/RobToPlc/Command/TelegramRobToPlcCommand
{attribute 'pack_mode' := '1'} 
// ------------------------------------------------------------------------- 
//  SRCI Robot Library                                                
// ------------------------------------------------------------------------- 
//                                                                           
//  Object:      TelegramPlcToRobMessage                                       
//  Author:      Thorsten Brach                                                
//  Date:        2024-11-02
//
//  Description:                                              
//   
//                                                                           
//  Copyright: 
//    (C) 2024 Thorsten Brach. All rights reserved                                                                                                                                            
//             Licensed under the LGPL-3.0 license.
//                                                                           
//  Disclaimer:                                                                           
//    This project is provided without any guarantee and can be used for   
//    private and commercial purposes. Any use is at the user’s 
//    own risk and responsibility.
//
// -------------------------------------------------------------------------
TYPE TelegramRobToPlcCommand :
STRUCT
  /// Header
  Header  : TelegramRobToPlcCommandHeader;
  /// Payload
  Payload : ARRAY[0..255] OF BYTE; // ToDo
END_STRUCT
END_TYPE

// Library/Structures/Telegram/RobToPlc/Command/TelegramRobToPlcCommandHeader
{attribute 'pack_mode' := '1'} 
// ------------------------------------------------------------------------- 
//  SRCI Robot Library                                                
// ------------------------------------------------------------------------- 
//                                                                           
//  Object:      TelegramPlcToRobMessageHeader                                       
//  Author:      Thorsten Brach                                                
//  Date:        2024-11-02
//
//  Description:                                              
//   
//                                                                           
//  Copyright: 
//    (C) 2024 Thorsten Brach. All rights reserved                                                                                                                                            
//             Licensed under the LGPL-3.0 license.
//                                                                           
//  Disclaimer:                                                                           
//    This project is provided without any guarantee and can be used for   
//    private and commercial purposes. Any use is at the user’s 
//    own risk and responsibility.
//
// -------------------------------------------------------------------------
TYPE TelegramRobToPlcCommandHeader :
STRUCT
  /// Parameter squence
  ParSeq               : BYTE;
  /// message Staet
  State                : CmdMessageState;
  /// Alarm Message Severity
  AlarmMessageSeverity : SINT;
  /// Alarm Message Code
  AlarmMessageCode     : UINT;
END_STRUCT
END_TYPE

// Library/Structures/Telegram/RobToPlc/CyclicOptional/Internal/TelegramRobToPlcCyclicOptionalCartesianPosition
{attribute 'pack_mode' := '1'} 
// ------------------------------------------------------------------------- 
//  SRCI Robot Library                                                
// ------------------------------------------------------------------------- 
//                                                                           
//  Object:      TelegramRobToPlcCyclicOptionalCartesianPosition                                       
//  Author:      Thorsten Brach                                                
//  Date:        2024-06-01
//
//  Description:                                              
//   
//                                                                           
//  Copyright: 
//    (C) 2024 Thorsten Brach. All rights reserved                                                                                                                                            
//             Licensed under the LGPL-3.0 license.
//                                                                           
//  Disclaimer:                                                                           
//    This project is provided without any guarantee and can be used for   
//    private and commercial purposes. Any use is at the user’s 
//    own risk and responsibility.
//
// -------------------------------------------------------------------------
TYPE TelegramRobToPlcCyclicOptionalCartesianPosition :
STRUCT
  /// TCP Position on the X-Axis
  X                    : REAL;
  /// TCP Position on the Y-Axis
  Y                    : REAL;
  /// TCP Position on the Z-Axis
  Z                    : REAL;
  /// Rotation around the X-Axis (RX)
  Rx                   : REAL;
  /// Rotation around the Y-Axis (RY)
  Ry                   : REAL;
  /// Rotation around the Z-Axis (RZ)
  Rz                   : REAL;
  /// Configuration
  Config               : WORD;
  /// Turns of J1 and J2
  Turns_J2_J1          : BYTE;
  /// Turns of J3 and J4
  Turns_J4_J3          : BYTE;
  /// Turns of J6 and J5
  Turns_J6_J5          : BYTE;
  /// Turns of E1
  Turns_E1             : BYTE;
  /// Position of first external axis
  E1                   : REAL;  
  /// Position of second external axis
  E2                   : REAL;
  /// Position of third external axis
  E3                   : REAL;
  /// Position of fourth external axis
  E4                   : REAL;
  /// Position of fifth external axis
  E5                   : REAL;
  /// Position of sixth external axis
  E6                   : REAL;      
  /// Tool Number
  ToolNo               : USINT;
  /// Frane Number
  FrameNo              : USINT;
  /// Currently used tool number
  CurrentlyUsedToolNo  : USINT;
  /// Currently used frame number
  CurrentlyUsedFrameNo : USINT;
  /// Reserve
  Reserve_1            : BYTE;
  /// Reserve
  Reserve_2            : BYTE;  
END_STRUCT
END_TYPE

// Library/Structures/Telegram/RobToPlc/CyclicOptional/Internal/TelegramRobToPlcCyclicOptionalCartesianPositionExt
{attribute 'pack_mode' := '1'} 
// ------------------------------------------------------------------------- 
//  SRCI Robot Library                                                
// ------------------------------------------------------------------------- 
//                                                                           
//  Object:      TelegramRobToPlcCyclicOptionalCartesianPosExt                                       
//  Author:      Thorsten Brach                                                
//  Date:        2024-06-01
//
//  Description:                                              
//   
//                                                                           
//  Copyright: 
//    (C) 2024 Thorsten Brach. All rights reserved                                                                                                                                            
//             Licensed under the LGPL-3.0 license.
//                                                                           
//  Disclaimer:                                                                           
//    This project is provided without any guarantee and can be used for   
//    private and commercial purposes. Any use is at the user’s 
//    own risk and responsibility.
//
// -------------------------------------------------------------------------
TYPE TelegramRobToPlcCyclicOptionalCartesianPositionExt :
STRUCT
  /// Position of second external axis
  E2 : REAL;
  /// Position of third external axis
  E3 : REAL;
  /// Position of fourth external axis
  E4 : REAL;
  /// Position of fifth external axis
  E5 : REAL;
  /// Position of sixth external axis
  E6 : REAL;    
END_STRUCT
END_TYPE

// Library/Structures/Telegram/RobToPlc/CyclicOptional/Internal/TelegramRobToPlcCyclicOptionalCurrent
{attribute 'pack_mode' := '1'} 
// ------------------------------------------------------------------------- 
//  SRCI Robot Library                                                
// ------------------------------------------------------------------------- 
//                                                                           
//  Object:      TelegramRobToPlcCyclicOptionalCurrent                                       
//  Author:      Thorsten Brach                                                
//  Date:        2024-06-01
//
//  Description:                                              
//   
//                                                                           
//  Copyright: 
//    (C) 2024 Thorsten Brach. All rights reserved                                                                                                                                            
//             Licensed under the LGPL-3.0 license.
//                                                                           
//  Disclaimer:                                                                           
//    This project is provided without any guarantee and can be used for   
//    private and commercial purposes. Any use is at the user’s 
//    own risk and responsibility.
//
// -------------------------------------------------------------------------
TYPE TelegramRobToPlcCyclicOptionalCurrent :
STRUCT
  /// Current of first joint of the robot
  J1 : REAL;
  /// Current of second joint of the robot
  J2 : REAL;
  /// Current of third joint of the robot
  J3 : REAL;
  /// Current of fourth joint of the robot
  J4 : REAL;
  /// Current of fifth joint of the robot
  J5 : REAL;
  /// Current of sixth joint of the robot
  J6 : REAL;  
END_STRUCT
END_TYPE

// Library/Structures/Telegram/RobToPlc/CyclicOptional/Internal/TelegramRobToPlcCyclicOptionalCurrentExt
{attribute 'pack_mode' := '1'} 
// ------------------------------------------------------------------------- 
//  SRCI Robot Library                                                
// ------------------------------------------------------------------------- 
//                                                                           
//  Object:      TelegramRobToPlcCyclicOptionalCurrentExt                                       
//  Author:      Thorsten Brach                                                
//  Date:        2024-06-01
//
//  Description:                                              
//   
//                                                                           
//  Copyright: 
//    (C) 2024 Thorsten Brach. All rights reserved                                                                                                                                            
//             Licensed under the LGPL-3.0 license.
//                                                                           
//  Disclaimer:                                                                           
//    This project is provided without any guarantee and can be used for   
//    private and commercial purposes. Any use is at the user’s 
//    own risk and responsibility.
//
// -------------------------------------------------------------------------
TYPE TelegramRobToPlcCyclicOptionalCurrentExt :
STRUCT
  /// Current of first external joint of the robot
  E1: REAL;
  /// Current of second external axis
  E2: REAL;
  /// Current of third external axis
  E3: REAL;
  /// Current of fourth external axis
  E4: REAL;
  /// Current of fifth external axis
  E5: REAL;
  /// Current of sixth external axis
  E6: REAL;  
END_STRUCT
END_TYPE

// Library/Structures/Telegram/RobToPlc/CyclicOptional/Internal/TelegramRobToPlcCyclicOptionalForce
{attribute 'pack_mode' := '1'} 
// ------------------------------------------------------------------------- 
//  SRCI Robot Library                                                
// ------------------------------------------------------------------------- 
//                                                                           
//  Object:      TelegramRobToPlcCyclicOptionalForce                                       
//  Author:      Thorsten Brach                                                
//  Date:        2024-06-01
//
//  Description:                                              
//   
//                                                                           
//  Copyright: 
//    (C) 2024 Thorsten Brach. All rights reserved                                                                                                                                            
//             Licensed under the LGPL-3.0 license.
//                                                                           
//  Disclaimer:                                                                           
//    This project is provided without any guarantee and can be used for   
//    private and commercial purposes. Any use is at the user’s 
//    own risk and responsibility.
//
// -------------------------------------------------------------------------
TYPE TelegramRobToPlcCyclicOptionalForce :
STRUCT
  /// Force on the X-Axis
  X : REAL;
  /// Force on the Y-Axis
  Y : REAL;
  /// Force on the Z-Axis
  Z : REAL;
  /// Force around the X-Axis (RX)
  Rx : REAL;
  /// Force around the Y-Axis (RY)
  Ry : REAL;
  /// Force around the Z-Axis (RZ)
  Rz : REAL;
END_STRUCT
END_TYPE

// Library/Structures/Telegram/RobToPlc/CyclicOptional/Internal/TelegramRobToPlcCyclicOptionalForceExt
{attribute 'pack_mode' := '1'} 
// ------------------------------------------------------------------------- 
//  SRCI Robot Library                                                
// ------------------------------------------------------------------------- 
//                                                                           
//  Object:      TelegramRobToPlcCyclicOptionalForceExt                                       
//  Author:      Thorsten Brach                                                
//  Date:        2024-06-01
//
//  Description:                                              
//   
//                                                                           
//  Copyright: 
//    (C) 2024 Thorsten Brach. All rights reserved                                                                                                                                            
//             Licensed under the LGPL-3.0 license.
//                                                                           
//  Disclaimer:                                                                           
//    This project is provided without any guarantee and can be used for   
//    private and commercial purposes. Any use is at the user’s 
//    own risk and responsibility.
//
// -------------------------------------------------------------------------
TYPE TelegramRobToPlcCyclicOptionalForceExt :
STRUCT
  /// Force on the external axis 1
  E1 : REAL;
  /// Force on the external axis 2
  E2 : REAL;
  /// Force on the external axis 3
  E3 : REAL;
  /// Force om the external axis 4
  E4 : REAL;
  /// Force on the external axis 5
  E5 : REAL;
  /// Force on the external axis 6
  E6 : REAL;
END_STRUCT
END_TYPE

// Library/Structures/Telegram/RobToPlc/CyclicOptional/Internal/TelegramRobToPlcCyclicOptionalJointPosition
{attribute 'pack_mode' := '1'} 
// ------------------------------------------------------------------------- 
//  SRCI Robot Library                                                
// ------------------------------------------------------------------------- 
//                                                                           
//  Object:      TelegramRobToPlcCyclicOptionalJointPosition                                       
//  Author:      Thorsten Brach                                                
//  Date:        2024-06-01
//
//  Description:                                              
//   
//                                                                           
//  Copyright: 
//    (C) 2024 Thorsten Brach. All rights reserved                                                                                                                                            
//             Licensed under the LGPL-3.0 license.
//                                                                           
//  Disclaimer:                                                                           
//    This project is provided without any guarantee and can be used for   
//    private and commercial purposes. Any use is at the user’s 
//    own risk and responsibility.
//
// -------------------------------------------------------------------------
TYPE TelegramRobToPlcCyclicOptionalJointPosition :
STRUCT
  /// Position of first joint of the robot
  J1 : REAL;
  /// Position of second joint of the robot
  J2 : REAL;
  /// Position of third joint of the robot
  J3 : REAL;
  /// Position of fourth joint of the robot
  J4 : REAL;
  /// Position of fifth joint of the robot
  J5 : REAL;
  /// Position of sixth joint of the robot
  J6 : REAL;
  /// Position of first external axis 
  E1 : REAL;  
  /// Reserve
  E1_Reserve : WORD;
END_STRUCT
END_TYPE

// Library/Structures/Telegram/RobToPlc/CyclicOptional/Internal/TelegramRobToPlcCyclicOptionalJointPositionExt
{attribute 'pack_mode' := '1'} 
// ------------------------------------------------------------------------- 
//  SRCI Robot Library                                                
// ------------------------------------------------------------------------- 
//                                                                           
//  Object:      TelegramRobToPlcCyclicOptionalJointPositionExt                                       
//  Author:      Thorsten Brach                                                
//  Date:        2024-06-01
//
//  Description:                                              
//   
//                                                                           
//  Copyright: 
//    (C) 2024 Thorsten Brach. All rights reserved                                                                                                                                            
//             Licensed under the LGPL-3.0 license.
//                                                                           
//  Disclaimer:                                                                           
//    This project is provided without any guarantee and can be used for   
//    private and commercial purposes. Any use is at the user’s 
//    own risk and responsibility.
//
// -------------------------------------------------------------------------
TYPE TelegramRobToPlcCyclicOptionalJointPositionExt :
STRUCT
  /// Position of second external axis
  E2: REAL;
  /// Position of third external axis
  E3: REAL;
  /// Position of fourth external axis
  E4: REAL;
  /// Position of fifth external axis
  E5: REAL;
  /// Position of sixth external axis
  E6: REAL;    
END_STRUCT
END_TYPE

// Library/Structures/Telegram/RobToPlc/CyclicOptional/Internal/TelegramRobToPlcCyclicOptionalSubProgramData
{attribute 'pack_mode' := '1'} 
// ------------------------------------------------------------------------- 
//  SRCI Robot Library                                                
// ------------------------------------------------------------------------- 
//                                                                           
//  Object:      TelegramRobToPlcCyclicOptionalSubProgramData                                       
//  Author:      Thorsten Brach                                                
//  Date:        2024-06-01
//
//  Description:                                              
//   
//                                                                           
//  Copyright: 
//    (C) 2024 Thorsten Brach. All rights reserved                                                                                                                                            
//             Licensed under the LGPL-3.0 license.
//                                                                           
//  Disclaimer:                                                                           
//    This project is provided without any guarantee and can be used for   
//    private and commercial purposes. Any use is at the user’s 
//    own risk and responsibility.
//
// -------------------------------------------------------------------------
TYPE TelegramRobToPlcCyclicOptionalSubProgramData :
STRUCT
  /// Sub program data
  Data : ARRAY [0..25] OF BYTE; {warning 'Add constant for DataMax'}
END_STRUCT
END_TYPE

// Library/Structures/Telegram/RobToPlc/CyclicOptional/TelegramRobToPlcCyclicOptionalData
{attribute 'pack_mode' := '1'} 
// ------------------------------------------------------------------------- 
//  SRCI Robot Library                                                
// ------------------------------------------------------------------------- 
//                                                                           
//  Object:      TelegramRobToPlcCyclicOptionalData                                       
//  Author:      Thorsten Brach                                                
//  Date:        2024-06-01
//
//  Description:                                              
//   
//                                                                           
//  Copyright: 
//    (C) 2024 Thorsten Brach. All rights reserved                                                                                                                                            
//             Licensed under the LGPL-3.0 license.
//                                                                           
//  Disclaimer:                                                                           
//    This project is provided without any guarantee and can be used for   
//    private and commercial purposes. Any use is at the user’s 
//    own risk and responsibility.
//
// -------------------------------------------------------------------------
TYPE TelegramRobToPlcCyclicOptionalData :
STRUCT
    /// Transmit cyclic data from PLC to RC for the usage in a subprogram on the RC called via the function “CallSubprogram”
  SubProgramData        :  TelegramRobToPlcCyclicOptionalSubProgramData;
  /// cartesian position with TCP position (X, Y,Z), rotation (RX, RY, RZ), configuration bytes (Config, TurnNumber), position of first external axis (E1) and corresponding coordinate systems (ToolNo, FrameNo)
  CartesianPosition     :  TelegramRobToPlcCyclicOptionalCartesianPosition;
  /// axes position with joint values (J1, J2, J3,J4, J5, J6) and position of first external axis (E1)
  JointPosition         :  TelegramRobToPlcCyclicOptionalJointPosition;
  /// force with the divided forces in the individual directions (X, Y, Z, RX, RY, RZ)
  Force                 :  TelegramRobToPlcCyclicOptionalForce;
  /// Transmit actual axes current of individual axes (J1, J2, J3, J4, J5, J6)
  Current               :  TelegramRobToPlcCyclicOptionalCurrent;
  /// Set to 1 to define two Sequences in one Telegram. If activated, 
  /// 2 sequences also has to be activated in the ClientServer direction.
  TwoSequences          : BYTE;  
  /// Transmit the external axis values for an extended cartesian position (E2, E3, E4, E5, E6)
  /// When selected, Tool and Frame will automatically cyclically be sent from client to server.
  CartesianPositionExt  :  TelegramRobToPlcCyclicOptionalCartesianPositionExt;
  /// Transmit the external axis values for an extended joint position (E2, E3, E4, E5, E6)
  JointPositionExt      :  TelegramRobToPlcCyclicOptionalJointPositionExt;
  /// Transmit actual axes force of individual axes (E1, E2, E3, E4, E5, E6)
  ForceExt              :  TelegramRobToPlcCyclicOptionalCurrentExt;
  /// Transmit actual axes current of individual axes (E1, E2, E3, E4, E5, E6)
  CurrentExt            :  TelegramRobToPlcCyclicOptionalCurrentExt;
END_STRUCT
END_TYPE

// Library/Structures/Telegram/RobToPlc/Footer/TelegramRobToPlcFooter
{attribute 'pack_mode' := '1'} 
// ------------------------------------------------------------------------- 
//  SRCI Robot Library                                                
// ------------------------------------------------------------------------- 
//                                                                           
//  Object:      TelegramPlcToRobFooter                                       
//  Author:      Thorsten Brach                                                
//  Date:        2024-06-01
//
//  Description:                                              
//   
//                                                                           
//  Copyright: 
//    (C) 2024 Thorsten Brach. All rights reserved                                                                                                                                            
//             Licensed under the LGPL-3.0 license.
//                                                                           
//  Disclaimer:                                                                           
//    This project is provided without any guarantee and can be used for   
//    private and commercial purposes. Any use is at the user’s 
//    own risk and responsibility.
//
// -------------------------------------------------------------------------
TYPE TelegramRobToPlcFooter :
STRUCT
  /// Reserve
  Reserve  : BYTE;
  /// Life Sign
  LifeSign : BYTE;
END_STRUCT
END_TYPE

// Library/Structures/Telegram/RobToPlc/Fragment/TelegramRobToPlcFragment
{attribute 'pack_mode' := '1'} 
// ------------------------------------------------------------------------- 
//  SRCI Robot Library                                                
// ------------------------------------------------------------------------- 
//                                                                           
//  Object:      TelegramPlcToRobFragment                                       
//  Author:      Thorsten Brach                                                
//  Date:        2024-11-02
//
//  Description:                                              
//   
//                                                                           
//  Copyright: 
//    (C) 2024 Thorsten Brach. All rights reserved                                                                                                                                            
//             Licensed under the LGPL-3.0 license.
//                                                                           
//  Disclaimer:                                                                           
//    This project is provided without any guarantee and can be used for   
//    private and commercial purposes. Any use is at the user’s 
//    own risk and responsibility.
//
// -------------------------------------------------------------------------
TYPE TelegramRobToPlcFragment :
STRUCT
  /// Header
  Header  : TelegramRobToPlcFragmentHeader;
  /// Command
  Command : TelegramRobToPlcCommand;
END_STRUCT
END_TYPE

// Library/Structures/Telegram/RobToPlc/Fragment/TelegramRobToPlcFragmentHeader
{attribute 'pack_mode' := '1'} 
// ------------------------------------------------------------------------- 
//  SRCI Robot Library                                                
// ------------------------------------------------------------------------- 
//                                                                           
//  Object:      TelegramPlcToRobFragmentHeader                                       
//  Author:      Thorsten Brach                                                
//  Date:        2024-11-02
//
//  Description:                                              
//   
//                                                                           
//  Copyright: 
//    (C) 2024 Thorsten Brach. All rights reserved                                                                                                                                            
//             Licensed under the LGPL-3.0 license.
//                                                                           
//  Disclaimer:                                                                           
//    This project is provided without any guarantee and can be used for   
//    private and commercial purposes. Any use is at the user’s 
//    own risk and responsibility.
//
// -------------------------------------------------------------------------
TYPE TelegramRobToPlcFragmentHeader :
STRUCT
  /// Command Instance Identifier used to assign the CMD payload to a specific CMD instance
  CmdID          : UINT;
  /// Empty reserve byte
  Reserve        : BYTE;
  /// Fragment Action Byte
  FragmentAction : BYTE;
  /// Append received payload in the receive buffer at this position
  PayloadPointer : UINT;
  /// Length of the CMD payload
  PayloadLength  : UINT;  
END_STRUCT
END_TYPE

// Library/Structures/Telegram/RobToPlc/Header/TelegramRobToPlcHeader
{attribute 'pack_mode' := '1'} 
// ------------------------------------------------------------------------- 
//  SRCI Robot Library                                                
// ------------------------------------------------------------------------- 
//                                                                           
//  Object:      TelegramRobToPlcCyclic                                       
//  Author:      Thorsten Brach                                                
//  Date:        2024-06-01
//
//  Description:                                              
//   
//                                                                           
//  Copyright: 
//    (C) 2024 Thorsten Brach. All rights reserved                                                                                                                                            
//             Licensed under the LGPL-3.0 license.
//                                                                           
//  Disclaimer:                                                                           
//    This project is provided without any guarantee and can be used for   
//    private and commercial purposes. Any use is at the user’s 
//    own risk and responsibility.
//
// -------------------------------------------------------------------------
TYPE TelegramRobToPlcHeader :
STRUCT
  /// Version of SRCI specification
  /// Bit 0-4 : Minor version = Features        (0..31)
  /// Bit 5-7 : Major version = Breaking change (0..07)
  SRCIVersion   : VersionStruct;
  /// Connection alive signal
  LifeSign      : BYTE;
  /// Reserved byte
  Reserved      : BYTE;
  /// Initialization and Telegram control state
  TelegramState : TelegramState;
  /// Combination of various RA related states.
  StatusRobotArm: DWORD;
  /// Actual override in percentage encoding 
  Override      : UINT;
END_STRUCT
END_TYPE

// Library/Structures/Telegram/RobToPlc/Sequence/TelegramRobToPlcSequence
{attribute 'pack_mode' := '1'} 
// ------------------------------------------------------------------------- 
//  SRCI Robot Library                                                
// ------------------------------------------------------------------------- 
//                                                                           
//  Object:      TelegramPlcToRobSequence                                       
//  Author:      Thorsten Brach                                                
//  Date:        2024-11-02
//
//  Description:                                              
//   
//                                                                           
//  Copyright: 
//    (C) 2024 Thorsten Brach. All rights reserved                                                                                                                                            
//             Licensed under the LGPL-3.0 license.
//                                                                           
//  Disclaimer:                                                                           
//    This project is provided without any guarantee and can be used for   
//    private and commercial purposes. Any use is at the user’s 
//    own risk and responsibility.
//
// -------------------------------------------------------------------------
TYPE TelegramRobToPlcSequence :
STRUCT
  /// Header
  Header   : TelegramRobToPlcSequenceHeader;
  /// Fragment
  Fragment : ARRAY[0..9] OF TelegramRobToPlcFragment;
END_STRUCT
END_TYPE

// Library/Structures/Telegram/RobToPlc/Sequence/TelegramRobToPlcSequenceHeader
{attribute 'pack_mode' := '1'} 
// ------------------------------------------------------------------------- 
//  SRCI Robot Library                                                
// ------------------------------------------------------------------------- 
//                                                                           
//  Object:      TelegramRobToPlcSequenceHeader                                       
//  Author:      Thorsten Brach                                                
//  Date:        2024-11-02
//
//  Description:                                              
//   
//                                                                           
//  Copyright: 
//    (C) 2024 Thorsten Brach. All rights reserved                                                                                                                                            
//             Licensed under the LGPL-3.0 license.
//                                                                           
//  Disclaimer:                                                                           
//    This project is provided without any guarantee and can be used for   
//    private and commercial purposes. Any use is at the user’s 
//    own risk and responsibility.
//
// -------------------------------------------------------------------------
TYPE TelegramRobToPlcSequenceHeader :
STRUCT
  /// Telegram Sequence and Acknowledgement number
  SEQ_ACK      : UINT;
  /// Length of the Telegram Sequence excluding this Telegram Sequence Header
  PayloadLength : UINT;
END_STRUCT
END_TYPE

// Library/Structures/Telegram/RobToPlc/TelegramRobToPlc
{attribute 'pack_mode' := '1'} 
// ------------------------------------------------------------------------- 
//  SRCI Robot Library                                                
// ------------------------------------------------------------------------- 
//                                                                           
//  Object:      TelegramRobToPlc                                       
//  Author:      Thorsten Brach                                                
//  Date:        2024-06-01
//
//  Description:                                              
//   
//                                                                           
//  Copyright: 
//    (C) 2024 Thorsten Brach. All rights reserved                                                                                                                                            
//             Licensed under the LGPL-3.0 license.
//                                                                           
//  Disclaimer:                                                                           
//    This project is provided without any guarantee and can be used for   
//    private and commercial purposes. Any use is at the user’s 
//    own risk and responsibility.
//
// -------------------------------------------------------------------------
TYPE TelegramRobToPlc :
STRUCT
  /// Telegram Header
  Header               : TelegramRobToPlcHeader;
  /// Cyclic optional data
  CyclicOptional       : TelegramRobToPlcCyclicOptionalData;
  /// Sequence Data
  Sequence             : ARRAY[0..1] OF TelegramRobToPlcSequence;
  /// Footer
  Footer               : TelegramRobToPlcFooter;
END_STRUCT
END_TYPE

// Library/Structures/Telegram/Telegram
{attribute 'pack_mode' := '1'} 
// ------------------------------------------------------------------------- 
//  SRCI Robot Library                                                
// ------------------------------------------------------------------------- 
//                                                                           
//  Object:      Telegram                                       
//  Author:      Thorsten Brach                                                
//  Date:        2024-06-01
//
//  Description:                                              
//   
//                                                                           
//  Copyright: 
//    (C) 2024 Thorsten Brach. All rights reserved                                                                                                                                            
//             Licensed under the LGPL-3.0 license.
//                                                                           
//  Disclaimer:                                                                           
//    This project is provided without any guarantee and can be used for   
//    private and commercial purposes. Any use is at the user’s 
//    own risk and responsibility.
//
// -------------------------------------------------------------------------
TYPE Telegram :
STRUCT
  /// PLC to Robot
  PlcToRob : TelegramPlcToRob;
  /// Robot to PLC
  RobToPlc : TelegramRobToPlc;
END_STRUCT
END_TYPE

